TYPE T_NOTT_CRYO_COOLDOWN_STAT :
STRUCT
	{attribute 'TcHmiSymbol.Show'}
	{attribute 'TcHmiSymbol.ReadOnly'}
	bEnabled:		BOOL := FALSE;	// Controller active while bEnable is TRUE
	bConfigured:	BOOL := FALSE;	// Flag if controller has been configured.
	bError:			BOOL;			// Flag if controller is OK
	{attribute 'TcHmiSymbol.Show'}
	{attribute 'TcHmiSymbol.ReadOnly'}
	bActive:		BOOL;			// Flag if controller is ACTIVE
	bWarning:		BOOL := FALSE;	// Flag if there is a warning
	bEmergency:		BOOL := FALSE;	// Flag if there was Emergency valve closure
	bPTC_On:		BOOL;			// Flag if Prevacuum Pump is running
	bPTC_Ready:		BOOL;			// Flag if Prevacuum Pump is Ready
	{attribute 'TcHmiSymbol.Show'}
	{attribute 'TcHmiSymbol.ReadOnly'}
	bAlarm:			BOOL;
	{attribute 'TcHmiSymbol.Show'}
	{attribute 'TcHmiSymbol.ReadOnly'}
	bPressureAlarm:	BOOL := FALSE;
	{attribute 'TcHmiSymbol.Show'}
	{attribute 'TcHmiSymbol.ReadOnly'}
	bPumpAlarm:		BOOL := FALSE;


	// Generic controller OK flag.
	// Used for problems other than from the actuator.
	// This flag is used for problems coming from controllers
	// that extend the functionality of FB_CRYO_BIN_CTRL.
	bCtrlOK:	BOOL := TRUE;		

	nState:			E_NOTT_CRYO_COOLDOWN_STATE := E_NOTT_CRYO_COOLDOWN_STATE.NONE;
	
	sErrorText:		STRING(64);		// Error as text
	sState:			STRING(64);		// State as text
	{attribute 'TcHmiSymbol.Show'}
	{attribute 'TcHmiSymbol.ReadOnly'}
	sStatus:		STRING(64);		// Status as text
END_STRUCT
END_TYPE

(* stored: Version 1.1.0.1, ProductVersion 3.1.4026.18
   DUT T_NOTT_CRYO_COOLDOWN_STAT: Id {07e7c200-faad-475b-b3d4-e6e35a89890e} *)
